{attribute 'strict'}
TYPE E_MachineCtrlStateInit :
(	
	(* Safety init *)
	MACHINE_STATE_INITIALIZING_MACHINE_LOGGER					:= 0,	(*  *)
	MACHINE_STATE_INITIALIZING_RECIPES_MANAGER						:= 10,	(*  *)
	MACHINE_STATE_INITIALIZING_CLEAR_ALL_ERRORS						:= 20,	(*  *)
	MACHINE_STATE_INITIALIZING_SAFETY_INITIALIZATION				:= 50,	(*  *)
	MACHINE_STATE_INITIALIZING_CHECK_ESTOP							:= 60,	(*  *)
	MACHINE_STATE_INITIALIZING_CHECK_DOOR_LOCKS						:= 80,	(*  *)
	MACHINE_STATE_INITIALIZING_ROBOTS_POWER_CHECK					:= 90,	(*  *)
	MACHINE_STATE_INITIALIZING_SAFETY_RESET							:= 100,	(*  *)
	MACHINE_STATE_INITIALIZING_SAFETY_START							:= 110,	(*  *)
	MACHINE_STATE_INITIALIZING_ROBOT_CONTROLERS_RESET				:= 120,	(*  *)
	MACHINE_STATE_INITIALIZING_SAFETY_CHECK							:= 130,	(*  *)
	MACHINE_STATE_INITIALIZING_ROBOT_AUTO_MODE_SW				:= 140,
	
	
	(* Robot init *)                                          		
	MACHINE_STATE_INITIALIZING_ROBOT_ABORT						:= 200,	(*  *)
	MACHINE_STATE_INITIALIZING_ROBOT_INIT						:= 210,	(*  *)
	MACHINE_STATE_INITIALIZING_ROBOT_HOME						:= 220,	(*  *)
	MACHINE_STATE_INITIALIZING_ROBOT_AUTOMATIC_MODE				:= 230,	(*  *)
	
	(* Rotary table init *)
	MACHINE_STATE_INITIALIZING_ROTARY_TABLE_ABORT				:= 400,
	MACHINE_STATE_INITIALIZING_ROTARY_TABLE_INIT				:= 410,	(*  *)
	MACHINE_STATE_INITIALIZING_ROTARY_TABLE_HOME				:= 420,	(*  *)

	(* Bowl feeder init *)
	MACHINE_STATE_INITIALIZING_BOWL_INIT						:= 500,

	MACHINE_STATE_INITIALIZING_DONE								:= 1000	(*  *)
)UINT;
END_TYPE

(* stored: Version 1.1.0.1, ProductVersion 3.1.4024.9
   DUT E_MachineCtrlStateInit: Id {031139da-8b48-4370-b379-8522fc5c6f57} *)
